FUNCTION_BLOCK FB_JsonLogger IMPLEMENTS I_Logger
VAR_INPUT
	eLogLevel:					E_Event;
	sFilePath:					STRING(255);
END_VAR
VAR_OUTPUT
END_VAR
VAR
	bExecute:			BOOL;
	jsonDoc:			SJsonValue;
	fbJson:				FB_JsonDynDomParser;

END_VAR

fbJson.LoadDocumentFromFile(sFilePath, bExecute);
fbJson.GetDocument()
fbJson.SaveDocumentToFile(sFilePath, bExecute);
fbJson.AddArrayMember(

METHOD M_Log
VAR_INPUT
	stEvent	: 		ST_Event;
END_VAR

VAR
	sMessage:			STRING(255);
END_VAR
IF stEvent.New THEN
	sMessage:= Concat(Concat(stEvent.Instance, ' | '), stEvent.Message);
	CASE stEvent.EventType OF
		E_Event.Error:
			ADSLOGSTR( msgCtrlMask := ADSLOG_MSGTYPE_ERROR , msgFmtStr := sMessage, strArg := '');
		E_Event.Warning:
			ADSLOGSTR( msgCtrlMask := ADSLOG_MSGTYPE_WARN , msgFmtStr := sMessage, strArg := '');
		E_Event.Information:
			ADSLOGSTR( msgCtrlMask := ADSLOG_MSGTYPE_HINT , msgFmtStr := sMessage, strArg := '');
		E_Event.Debug:
			ADSLOGSTR( msgCtrlMask := ADSLOG_MSGTYPE_HINT, msgFmtStr := sMessage, strArg := '');
		E_Event.Verbose:
			ADSLOGSTR( msgCtrlMask := ADSLOG_MSGTYPE_HINT , msgFmtStr := sMessage, strArg := '');
	END_CASE
END_IF
END_METHOD

END_FUNCTION_BLOCK

(* stored: Version 1.1.0.1, ProductVersion 3.1.4024.12
   POU FB_JsonLogger: Id {b9ff5c72-49fc-000f-0b8a-0489330fd727}, SpecialFunc None
   Method M_Log: Id {6b0311b7-02e1-0a93-0f6f-4a3bfbdf6fcf} *)
